// TwinCAT 3 PLC project Controller
// Title: test
// Company: test
// Author: test
// ProjectVersion: 1.0
// Description: test
// ProgramVersion: 3.1.4026.1+c9eadab3edd020c56c333d811d5b3c408c2550c8
// CompilerDefines: test
// libraries:
//   Tc2_Standard, * (Beckhoff Automation GmbH)
//   Tc2_System, * (Beckhoff Automation GmbH)
// project tree:
//   / MAIN.TcPOU, PidController.TcPOU, PidControllerTest.TcPOU, PlcTask.TcTTO

CONFIGURATION Controller
    RESOURCE PLC ON TwinCAT3
        TASK PlcTask(INTERVAL := T#200us, PRIORITY := 20);
        PROGRAM MAIN WITH PlcTask : MAIN;
    END_RESOURCE
END_CONFIGURATION

// ---- MAIN.TcPOU

PROGRAM MAIN
VAR
	testPid_ : BOOL := FALSE;
	testController_ : PidControllerTest;
END_VAR


IF testPid_ THEN
	testController_.cyclic();
ELSE
	testController_.reset();
END_IF

END_PROGRAM

// ---- PidControllerTest.TcPOU

FUNCTION_BLOCK PidControllerTest
VAR
	actualValuePid_ : LREAL := 5;
	controlOutputPid_ : LREAL;
	controller_ : PidController(desiredValue:=20, kp:=0.5, ki:=0.01, kd:=0.1);
END_VAR


METHOD cyclic

controlOutputPid_ := controller_.cyclic(actualValuePid_);

IF 	  controlOutputPid_ >= 5 THEN actualValuePid_ := actualValuePid_ + 0.1;
ELSIF controlOutputPid_ >= 6 THEN actualValuePid_ := actualValuePid_ + 0.2;
ELSIF controlOutputPid_ >= 7 THEN actualValuePid_ := actualValuePid_ + 0.3;
ELSIF controlOutputPid_ >= 8 THEN actualValuePid_ := actualValuePid_ + 0.4;
ELSIF controlOutputPid_ >= 9 THEN actualValuePid_ := actualValuePid_ + 0.5;
	
ELSIF controlOutputPid_ <= 5 THEN actualValuePid_ := actualValuePid_ - 0.1;
ELSIF controlOutputPid_ <= 4 THEN actualValuePid_ := actualValuePid_ - 0.2;
ELSIF controlOutputPid_ <= 3 THEN actualValuePid_ := actualValuePid_ - 0.3;
ELSIF controlOutputPid_ <= 2 THEN actualValuePid_ := actualValuePid_ - 0.4;
ELSIF controlOutputPid_ <= 1 THEN actualValuePid_ := actualValuePid_ - 0.5;
END_IF
END_METHOD


METHOD reset

controller_.reset();
END_METHOD

END_FUNCTION_BLOCK

// ---- PidController.TcPOU

FUNCTION_BLOCK PidController
VAR
	desiredValue_ : LREAL;
	actualValue_ : LREAL;
	previousValue_ : LREAL;
	error_ : LREAL;
	controlOutput_ : LREAL;
	
	cycleTime_ : UDINT;
	
	firstLoop_ : BOOL := TRUE;
	
	kp_ : LREAL;
	ki_ : LREAL;
	kd_ : LREAL;
	
	p_ : LREAL;
	i_ : LREAL;
	d_ : LREAL;
END_VAR


METHOD calculateDifferential

d_ := kd_ * ((actualValue_ - previousValue_) / cycleTime_);

IF previousValue_ = 0 THEN
	d_ := 0;
END_IF

previousValue_ := actualValue_;
END_METHOD


METHOD calculateIntegral

i_ := i_ + ki_ * error_;
END_METHOD


METHOD calculateOutput : LREAL

calculateOutput := p_ + i_ + d_;
END_METHOD


METHOD calculateProportional

p_ := kp_ * error_;
END_METHOD


METHOD cyclic
VAR_INPUT
	actualValue : LREAL;
END_VAR
VAR_OUTPUT
	controlOutput : LREAL;
END_VAR

IF firstLoop_ THEN
	getCycleTime();
	firstLoop_ := FALSE;
END_IF

actualValue_ := actualValue;
error_ := desiredValue_ - actualValue_;

// P
calculateProportional();
// I
calculateIntegral();
// D 
calculateProportional();

controlOutput := calculateOutput();
END_METHOD

//FB_Init is always available implicitly and it is used primarily for initialization.
//The return value is not evaluated. For a specific influence, you can also declare the
//methods explicitly and provide additional code there with the standard initialization
//code. You can evaluate the return value.
METHOD FB_Init: BOOL
VAR_INPUT
    bInitRetains: BOOL; // TRUE: the retain variables are initialized (reset warm / reset cold)
    bInCopyCode: BOOL;  // TRUE: the instance will be copied to the copy code afterward (online change)
		desiredValue : LREAL;
		kp : LREAL;
		ki : LREAL;
		kd : LREAL;
END_VAR

desiredValue_ := desiredValue;
kp_ := kp;
ki_ := ki;
kd_ := kd;
END_METHOD


METHOD getCycleTime
VAR
	taskIndex : DINT;
END_VAR

taskIndex := Tc2_System.GETCURTASKINDEXEX();
IF taskIndex > 0 THEN
    cycleTime_ := TwinCAT_SystemInfoVarList._TaskInfo[taskIndex].CycleTime;
END_IF
END_METHOD


METHOD reset

actualValue_ := 0;
previousValue_ := 0;
error_ := 0;
controlOutput_ := 0;
cycleTime_ := 0;
firstLoop_ := TRUE;
p_ := 0;
i_ := 0;
d_ := 0;
END_METHOD

END_FUNCTION_BLOCK
